RoboDK station: Kawasaki.rdk

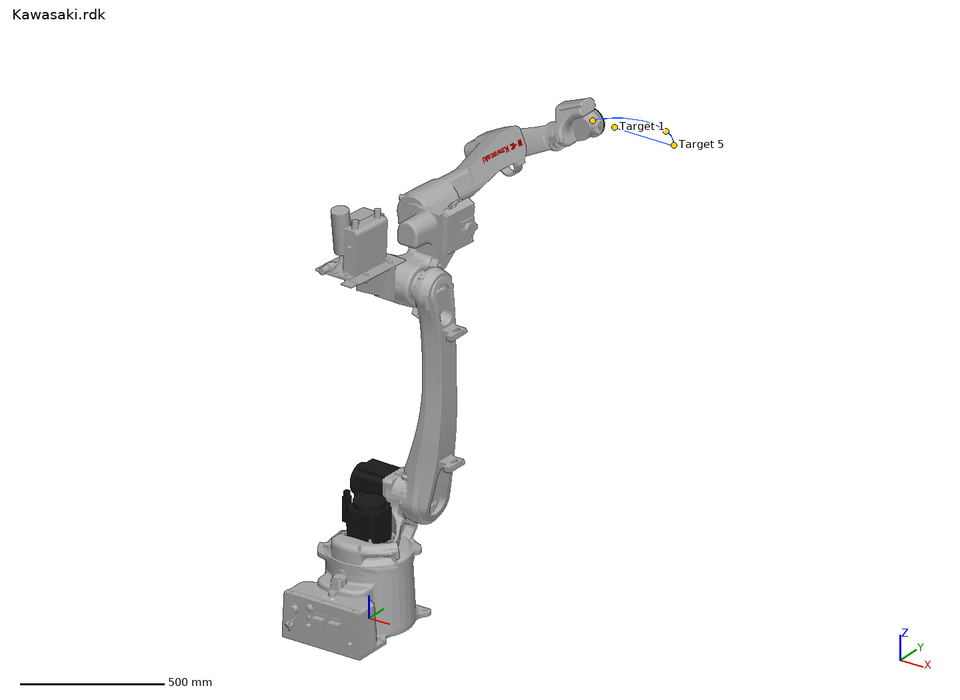
[picture v0: the station drawn from its stored meshes, robots at their saved joint values, targets as dots, program paths as lines]
Station Kawasaki. Poses are relative to the parent item; angles as X-Y-Z fixed-axis rotations.
  - frame Kawasaki BA006L Base at (0, 0, 0) mm
    - robot Kawasaki BA006L: 6 axes, payload 6 kg, reach 2036 mm, repeatability 0.08 mm, weight 160 kg
        modified DH rows (alpha deg, a mm, theta deg, d mm): 0, 0, 0, 430; -90, 165, -90, 0; 0, 820, -90, 0; -90, 210, 0, 1030; 90, 0, 0, 0; -90, 0, 180, 115
        base shift (0, 0, 0) mm, rotated rx 0 ry 0 rz 90 deg
        joint limits [-165, -90, -155, -180, -135, -360] to [165, 150, 135, 180, 135, 360]; home [0, 0, -90, 0, 0, 0]; saved at [1.365, -0.648, -93.662, 155.614, -3.308, -155.65]
    - target Target 1 (Cartesian target) at (123.18, 1310, 1405.5) mm, rotated rx -90 ry 0 rz 0 deg; joints [5.885, -0.23, -93.246, 117.043, -6.611, -117.198] of Kawasaki BA006L
    - target Target 5 (Cartesian target) at (372.97, 1310, 1405.5) mm, rotated rx -90 ry 0 rz 0 deg; joints [17.334, 3.316, -89.625, 99.335, -17.574, -99.783] of Kawasaki BA006L
    - target Target 3 (Cartesian target) at (285.5, 1388.79, 1405.5) mm, rotated rx -90 ry 0 rz 0 deg; joints [12.633, 7.127, -85.54, 101.729, -12.907, -102.025] of Kawasaki BA006L
    - target Target 4 (Cartesian target) at (28.48, 1310, 1405.5) mm, rotated rx -90 ry 0 rz 0 deg; joints [1.365, -0.648, -93.662, 155.614, -3.308, -155.65] of Kawasaki BA006L
  - program Prog1 (4 instructions, listed below)
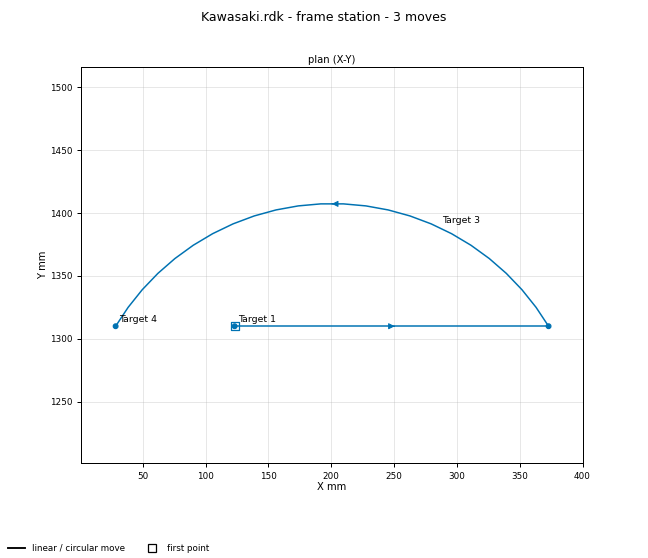
[picture p0: tool path of Kawasaki.rdk in frame station, 3 of 3 moves have a stored position in this frame; points joined in program order, loops and branches not executed]

--- program Prog1 (robot Kawasaki BA006L) ---
  Set Ref.: Kawasaki BA006L Base
  MoveJ (Target 1)
  MoveL (Target 5)
  MoveC (Target 3, Target 4)
